FUNCTION_BLOCK CentralServer (* Composite Function Block Type that operates using Central Server *)
  (* Standard: 61499-2 *)
  (* Version 0.2, 2003-12-05, JHC, Rockwell Automation, Renamed from NEWCOMPFB. *)
  (* Version 0.1, 2002-01-08, JHC, Rockwell Automation, Added DLY FB as example. *)
  (* Version 0.0, 2000-05-27, JHC, Rockwell Automation *)
  (* Compiler header: package fb.rt.cs725; *)
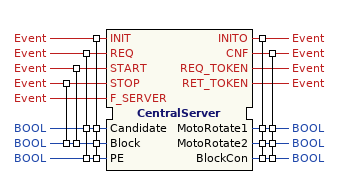
  EVENT_INPUT
    INIT WITH Candidate, Block, PE; (* Initialization Request *)
    REQ WITH Candidate, PE; (* Normal Execution Request *)
    START WITH Block;
    STOP WITH Block;
    F_SERVER;
  END_EVENT
  EVENT_OUTPUT
    INITO WITH MotoRotate1, MotoRotate2, BlockCon; (* Initialization Confirm *)
    CNF WITH MotoRotate1, MotoRotate2, BlockCon; (* Execution Confirmation *)
    REQ_TOKEN;
    RET_TOKEN;
  END_EVENT
  VAR_INPUT
    Candidate : BOOL;
    Block : BOOL;
    PE : BOOL;
  END_VAR
  VAR_OUTPUT
    MotoRotate1 : BOOL;
    MotoRotate2 : BOOL;
    BlockCon : BOOL;
  END_VAR
  FBS
    FC11 : ConveyorCTL(PE := 0, Block := 0, Candidate := 0);
    Conveyor2 : CentralServerClient;
  END_FBS
  EVENT_CONNECTIONS
    INIT TO FC11.INIT;
    STOP TO Conveyor2.CAS_STOP;
    START TO Conveyor2.CAS_START;
    REQ TO Conveyor2.REQ;
    Conveyor2.CNF TO CNF;
    Conveyor2.INITO TO INITO;
    FC11.INITO TO Conveyor2.INIT;
    Conveyor2.STOP TO FC11.CAS_STOP;
    Conveyor2.START TO FC11.CAS_START;
    Conveyor2.REQ_TOKEN TO REQ_TOKEN;
    Conveyor2.RET_TOKEN TO RET_TOKEN;
    F_SERVER TO Conveyor2.F_SERVER;
    REQ TO FC11.REQ;
  END_CONNECTIONS
  DATA_CONNECTIONS
    FC11.MotoRotate TO MotoRotate1;
    PE TO Conveyor2.PE;
    Block TO Conveyor2.Block;
    Candidate TO Conveyor2.Candidate;
    Conveyor2.MotoRotate TO MotoRotate2;
    Conveyor2.BlockCon TO BlockCon;
  END_CONNECTIONS
END_FUNCTION_BLOCK
